// TIA Portal V20 export
FUNCTION_BLOCK "FB_Search_Water_Foutain"   // FB9, LAD
{ S7_Optimized_Access := 'TRUE' }
// stored: MemoryReserve 100, SetENOAutomatically false
   VAR_INPUT
      Trigger_Read_Serial_Number_Exit_Functional_Test : Bool;
      Serial_Number : String[17];
      Functional_Tests_Panels : Array[0..31] of "Functional_Test";
   END_VAR
   VAR_OUTPUT
      Found_Functional_Test : Bool;
      Water_Foutain_Fail_Functional_Test : Bool;
      DataLog_Write : Bool;
      i : SInt;
      Search_Functional_Test : "Functional_Test";
      Reset_PLC_Functional_Test : Array[0..31] of Bool;
   END_VAR
   VAR
      Timer_Delay_Write_DataLog { S7_SetPoint := 'True'} : TON_TIME;
   END_VAR
   // Functional_Tests_Panels[0].Panel_Number := 0;
   // Functional_Tests_Panels[1].Panel_Number := 1;
   // Functional_Tests_Panels[2].Panel_Number := 2;
   // Functional_Tests_Panels[3].Panel_Number := 3;
   // Functional_Tests_Panels[4].Panel_Number := 4;
   // Functional_Tests_Panels[5].Panel_Number := 5;
   // Functional_Tests_Panels[6].Panel_Number := 6;
   // Functional_Tests_Panels[7].Panel_Number := 7;
   // Functional_Tests_Panels[8].Panel_Number := 8;
   // Functional_Tests_Panels[9].Panel_Number := 9;
   // Functional_Tests_Panels[10].Panel_Number := 10;
   // Functional_Tests_Panels[11].Panel_Number := 11;
   // Functional_Tests_Panels[12].Panel_Number := 12;
   // Functional_Tests_Panels[13].Panel_Number := 13;
   // Functional_Tests_Panels[14].Panel_Number := 14;
   // Functional_Tests_Panels[15].Panel_Number := 15;
   // Functional_Tests_Panels[16].Panel_Number := 16;
   // Functional_Tests_Panels[17].Panel_Number := 17;
   // Functional_Tests_Panels[18].Panel_Number := 18;
   // Functional_Tests_Panels[19].Panel_Number := 19;
   // Functional_Tests_Panels[20].Panel_Number := 20;
   // Functional_Tests_Panels[21].Panel_Number := 21;
   // Functional_Tests_Panels[22].Panel_Number := 22;
   // Functional_Tests_Panels[23].Panel_Number := 23;
   // Functional_Tests_Panels[24].Panel_Number := 24;
   // Functional_Tests_Panels[25].Panel_Number := 25;
   // Functional_Tests_Panels[26].Panel_Number := 26;
   // Functional_Tests_Panels[27].Panel_Number := 27;
   // Functional_Tests_Panels[28].Panel_Number := 28;
   // Functional_Tests_Panels[29].Panel_Number := 29;
   // Functional_Tests_Panels[30].Panel_Number := 30;
   // Functional_Tests_Panels[31].Panel_Number := 31;
   VAR_TEMP   // added for the SCL form of the ladder/FBD networks
      _w1 : Bool;
   END_VAR
BEGIN

REGION Network 1
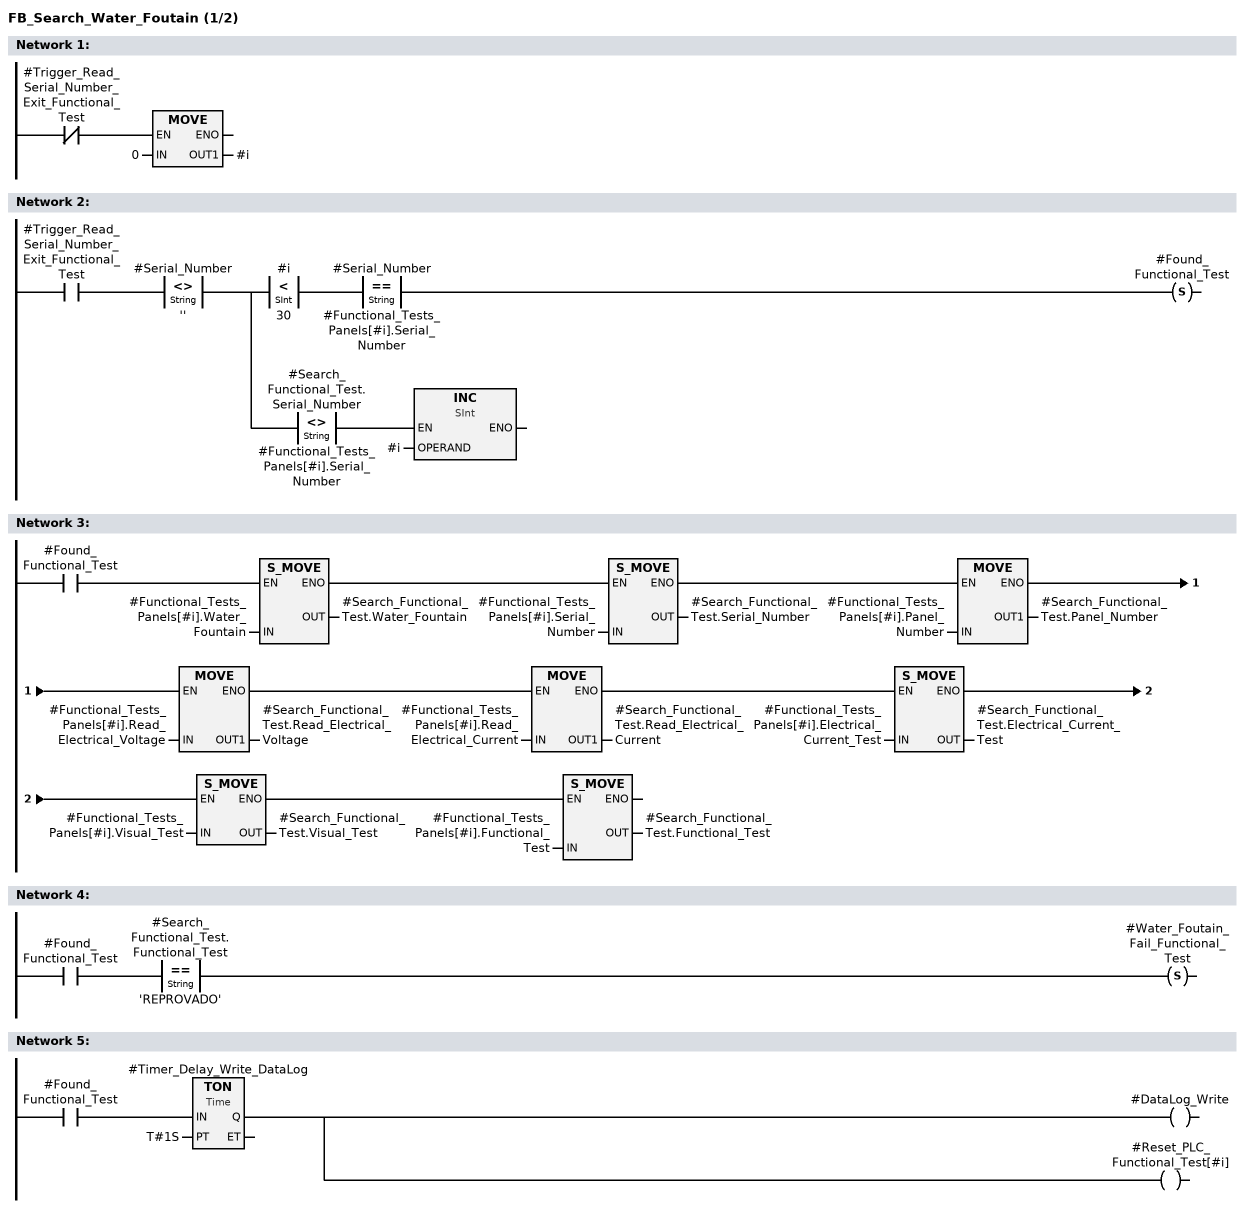
   RUNG wire#powerrail
      I_Contact( #Trigger_Read_Serial_Number_Exit_Functional_Test )
      Move(in := 0, out1 => #i)
   END_RUNG
   // the same network as SCL:
   IF NOT #Trigger_Read_Serial_Number_Exit_Functional_Test THEN #i := 0; END_IF;
END_REGION

REGION Network 2
   RUNG wire#powerrail
      Contact( #Trigger_Read_Serial_Number_Exit_Functional_Test )
      { S7_Templates := "SrcType := String" } NE_Contact(in1 := #Serial_Number, in2 := '')
      wire#w1
      { S7_Templates := "SrcType := SInt" } LT_Contact(in1 := #i, in2 := 30)
      { S7_Templates := "SrcType := String" } EQ_Contact(in1 := #Serial_Number, in2 := #Functional_Tests_Panels[#i].Serial_Number)
      S_Coil( #Found_Functional_Test )
   END_RUNG
   RUNG wire#w1
      { S7_Templates := "SrcType := String" } NE_Contact(in1 := #Search_Functional_Test.Serial_Number, in2 := #Functional_Tests_Panels[#i].Serial_Number)
      { S7_Templates := "DestType := SInt" } Inc( #i )
   END_RUNG
   // the same network as SCL:
   #_w1 := #Trigger_Read_Serial_Number_Exit_Functional_Test AND (#Serial_Number <> '');
   IF #_w1 AND (#i < 30) AND (#Serial_Number = #Functional_Tests_Panels[#i].Serial_Number) THEN
       #Found_Functional_Test := TRUE;
   END_IF;
   IF #_w1 AND (#Search_Functional_Test.Serial_Number <> #Functional_Tests_Panels[#i].Serial_Number) THEN
       #i := #i + 1;
   END_IF;
END_REGION

REGION Network 3
   RUNG wire#powerrail
      Contact( #Found_Functional_Test )
      S_Move(in := #Functional_Tests_Panels[#i].Water_Fountain, out => #Search_Functional_Test.Water_Fountain)
      S_Move(in := #Functional_Tests_Panels[#i].Serial_Number, out => #Search_Functional_Test.Serial_Number)
      Move(in := #Functional_Tests_Panels[#i].Panel_Number, out1 => #Search_Functional_Test.Panel_Number)
      Move(in := #Functional_Tests_Panels[#i].Read_Electrical_Voltage, out1 => #Search_Functional_Test.Read_Electrical_Voltage)
      Move(in := #Functional_Tests_Panels[#i].Read_Electrical_Current, out1 => #Search_Functional_Test.Read_Electrical_Current)
      S_Move(in := #Functional_Tests_Panels[#i].Electrical_Current_Test, out => #Search_Functional_Test.Electrical_Current_Test)
      S_Move(in := #Functional_Tests_Panels[#i].Visual_Test, out => #Search_Functional_Test.Visual_Test)
      S_Move(in := #Functional_Tests_Panels[#i].Functional_Test, out => #Search_Functional_Test.Functional_Test)
   END_RUNG
   // the same network as SCL:
   IF #Found_Functional_Test THEN
       #Search_Functional_Test.Water_Fountain := #Functional_Tests_Panels[#i].Water_Fountain;
       #Search_Functional_Test.Serial_Number := #Functional_Tests_Panels[#i].Serial_Number;
       #Search_Functional_Test.Panel_Number := #Functional_Tests_Panels[#i].Panel_Number;
       #Search_Functional_Test.Read_Electrical_Voltage := #Functional_Tests_Panels[#i].Read_Electrical_Voltage;
       #Search_Functional_Test.Read_Electrical_Current := #Functional_Tests_Panels[#i].Read_Electrical_Current;
       #Search_Functional_Test.Electrical_Current_Test := #Functional_Tests_Panels[#i].Electrical_Current_Test;
       #Search_Functional_Test.Visual_Test := #Functional_Tests_Panels[#i].Visual_Test;
       #Search_Functional_Test.Functional_Test := #Functional_Tests_Panels[#i].Functional_Test;
   END_IF;
END_REGION

REGION Network 4
   RUNG wire#powerrail
      Contact( #Found_Functional_Test )
      { S7_Templates := "SrcType := String" } EQ_Contact(in1 := #Search_Functional_Test.Functional_Test, in2 := 'REPROVADO')
      S_Coil( #Water_Foutain_Fail_Functional_Test )
   END_RUNG
   // the same network as SCL:
   IF #Found_Functional_Test AND (#Search_Functional_Test.Functional_Test = 'REPROVADO') THEN
       #Water_Foutain_Fail_Functional_Test := TRUE;
   END_IF;
END_REGION

REGION Network 5
   RUNG wire#powerrail
      Contact( #Found_Functional_Test )
      { S7_Templates := "time_type := Time" } #Timer_Delay_Write_DataLog.TON(pt := T#1S, et =>)
      wire#w1
      Coil( #DataLog_Write )
   END_RUNG
   RUNG wire#w1
      Coil( #Reset_PLC_Functional_Test[#i] )
   END_RUNG
   // the same network as SCL:
   #Timer_Delay_Write_DataLog(IN := #Found_Functional_Test, PT := T#1S);   // TON
   #DataLog_Write := #Timer_Delay_Write_DataLog.Q;
   #Reset_PLC_Functional_Test[#i] := #Timer_Delay_Write_DataLog.Q;
END_REGION

REGION Network 6
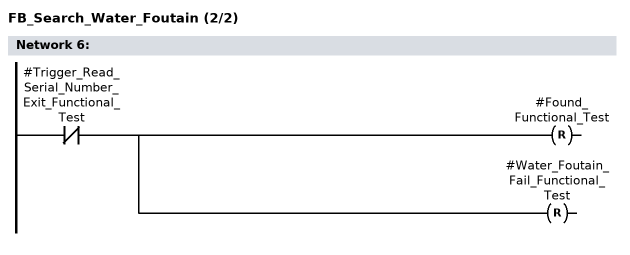
   RUNG wire#powerrail
      I_Contact( #Trigger_Read_Serial_Number_Exit_Functional_Test )
      wire#w1
      R_Coil( #Found_Functional_Test )
   END_RUNG
   RUNG wire#w1
      R_Coil( #Water_Foutain_Fail_Functional_Test )
   END_RUNG
   // the same network as SCL:
   IF NOT #Trigger_Read_Serial_Number_Exit_Functional_Test THEN
       #Found_Functional_Test := FALSE;
       #Water_Foutain_Fail_Functional_Test := FALSE;
   END_IF;
END_REGION
END_FUNCTION_BLOCK
